FUNCTION F_CtoF : LREAL
VAR_INPUT
	lrTempInC : LREAL;
END_VAR
VAR
END_VAR

F_CtoF := lrTempInC * (9.0/5.0) + 32.0;

END_FUNCTION

(* stored: Version 1.1.0.1, ProductVersion 3.1.4024.9
   POU F_CtoF: Id {d3017ad7-e8df-4ce9-be86-335e073c1cc9}, SpecialFunc None *)
